SUBAPPLICATION Uebung_020e2 (* DigitalInput_I1 auf DigitalOutput_Q1; FB_TOF; Ausschaltverzögert *)
  (* Standard: 61499-2; Description: Copyright (c) 2023 Meisterschulen am Ostbahnhof This program and the accompanying materials are made available under the terms of the Eclipse Public License 2.0 which is available at https://www.eclipse.org/legal/epl-2.0/ SPDX-License-Identifier: EPL-2.0 *)
  (* Version 1.0, 2023-10-23, Franz Höpfinger, Meisterschulen am Ostbahnhof *)
  IMPORT logiBUS::io::DI::logiBUS_DI::Input_I1;
  IMPORT logiBUS::io::DQ::logiBUS_DO::Output_Q1;
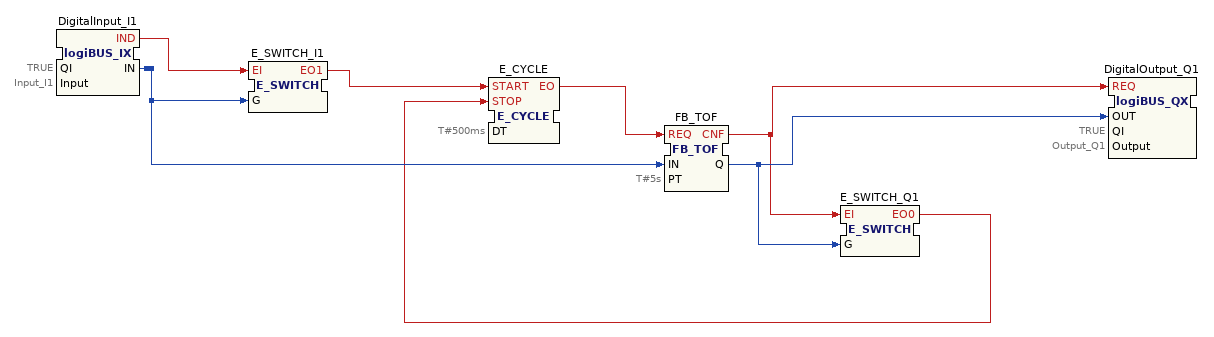
  (* E_CYCLE bestimmt, wie oft FB_TOF den ET aktualisert *)
  FBS
    DigitalOutput_Q1 : logiBUS::io::DQ::logiBUS_QX(QI := TRUE, Output := Output_Q1);
    DigitalInput_I1 : logiBUS::io::DI::logiBUS_IX(QI := TRUE, Input := Input_I1);
    FB_TOF : iec61131::timers::FB_TOF(PT := T#5s);
    E_CYCLE : iec61499::events::E_CYCLE(DT := T#500ms);
    E_SWITCH_I1 : iec61499::events::E_SWITCH;
    E_SWITCH_Q1 : iec61499::events::E_SWITCH;
  END_FBS
  EVENT_CONNECTIONS
    FB_TOF.CNF TO DigitalOutput_Q1.REQ;
    E_SWITCH_I1.EO1 TO E_CYCLE.START;
    DigitalInput_I1.IND TO E_SWITCH_I1.EI;
    E_CYCLE.EO TO FB_TOF.REQ;
    FB_TOF.CNF TO E_SWITCH_Q1.EI;
    E_SWITCH_Q1.EO0 TO E_CYCLE.STOP;
  END_CONNECTIONS
  DATA_CONNECTIONS
    DigitalInput_I1.IN TO FB_TOF.IN;
    FB_TOF.Q TO DigitalOutput_Q1.OUT;
    DigitalInput_I1.IN TO E_SWITCH_I1.G;
    FB_TOF.Q TO E_SWITCH_Q1.G;
  END_CONNECTIONS
END_SUBAPPLICATION
